FUNCTION_BLOCK AXE_plant_FV
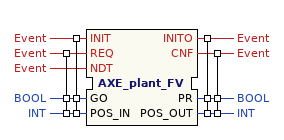
  EVENT_INPUT
    INIT WITH GO, POS_IN;
    REQ WITH GO, POS_IN;
    NDT;
  END_EVENT
  EVENT_OUTPUT
    INITO WITH PR, POS_OUT;
    CNF WITH PR, POS_OUT;
  END_EVENT
  VAR_INPUT
    GO : BOOL;
    POS_IN : INT;
  END_VAR
  VAR_OUTPUT
    PR : BOOL;
    POS_OUT : INT;
  END_VAR
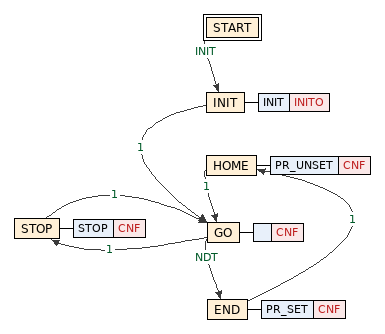
  EC_STATES
    START;
    HOME : PR_UNSET -> CNF;
    GO : -> CNF;
    END : PR_SET -> CNF;
    STOP : STOP -> CNF;
    INIT : INIT -> INITO;
  END_STATES
  EC_TRANSITIONS
    HOME TO GO := 1;
    STOP TO GO := 1;
    GO TO STOP := 1;
    GO TO END := NDT;
    END TO HOME := 1;
    START TO INIT := INIT;
    INIT TO GO := 1;
  END_TRANSITIONS
  ALGORITHM INIT IN ST:
PR := FALSE;&#38;#10;
  END_ALGORITHM
  ALGORITHM PR_SET IN ST:
PR := TRUE;&#38;#10;POS_OUT := POS_IN;&#38;#10;
  END_ALGORITHM
  ALGORITHM STOP IN ST:
PR := FALSE;&#38;#10;POS_OUT := 5;&#38;#10;
  END_ALGORITHM
  ALGORITHM PR_UNSET IN ST:
PR := FALSE;&#38;#10;
  END_ALGORITHM
END_FUNCTION_BLOCK
